Fanuc KAREL source: CALL_PROGLIN.kl

PROGRAM T
%NOLOCKGROUP
VAR
 v0 : STRING[40]
 v1 : INTEGER
 v2 : INTEGER
 v3 : BOOLEAN
BEGIN
 CALL_PROGLIN(v0, v1, v2, v3)
END T
